Staubli VAL3: SimpleMessage.pjx

--- SimpleMessage.pjx ---
Parameters version=s7.3 stackSize=5000 millimeterUnit=true
Data file=SimpleMessage.dtx
Type name=CommType path=Disk://CommType/CommType.pjx
Type name=ReplyType path=Disk://ReplyType/ReplyType.pjx

--- SimpleMessage.dtx ---
public CommType commType
  [0]
    num nRequest = 2
    num nResponse = 3
public ReplyType replyType
  [0]
    num nSuccess = 1
    num nFailure = 2
